{attribute 'GeneratedUsingTerminal: ELM2644-0000-0016'}
{attribute addProperty BoxType "ELM2644-0000-0016"}
{attribute addProperty Description "ELM2644 4Ch. Multiplexer Ausgang 1x4 Reed-Relais 48V AC/DC, 1A, potential-free"}
{attribute addProperty Physics "KK"}
{attribute addProperty Id "DO_Inputs_DeviceAT %I*DO_Inputs_Device_4A9049C53DO_Group_1_OutputsAT %Q*DO_Group_1_Outputs_07009A9C4DO_Group_2_OutputsAT %Q*DO_Group_2_Outputs_3033EF654DO_Group_3_OutputsAT %Q*DO_Group_3_Outputs_22DD3C324DO_Group_4_OutputsAT %Q*DO_Group_4_Outputs_5E5504974WcStateAT %I*WcState_9091E0EB2InfoDataAT %I*InfoData_BEF6B88E18"}
{attribute addProperty CRC "2656463402"}
{attribute addProperty Size "39"}
TYPE ELM2644_9E566A2A EXTENDS EtcSlaveTerminalBase_947E5A46 :
STRUCT
	{attribute addProperty Name "DO_Inputs_Device"}
	DO_Inputs_Device : DO_Inputs_Device_4A9049C5;
	{attribute addProperty Name "DO_Group_1_Outputs"}
	DO_Group_1_Outputs : DO_Group_1_Outputs_07009A9C;
	{attribute addProperty Name "DO_Group_2_Outputs"}
	DO_Group_2_Outputs : DO_Group_2_Outputs_3033EF65;
	{attribute addProperty Name "DO_Group_3_Outputs"}
	DO_Group_3_Outputs : DO_Group_3_Outputs_22DD3C32;
	{attribute addProperty Name "DO_Group_4_Outputs"}
	DO_Group_4_Outputs : DO_Group_4_Outputs_5E550497;
	{attribute addProperty Name "WcState"}
	WcState : WcState_9091E0EB;
	{attribute addProperty Name "InfoData"}
	InfoData : InfoData_BEF6B88E;
END_STRUCT
END_TYPE

(* stored: Version 1.2.0.0, ProductVersion 3.1.4024.9
   DUT ELM2644_9E566A2A: Id {1eec9f3b-bce1-4564-9827-77053e9958af} *)
